ADAPTER WagoBusAdapter
  (* Standard: 61499-2; Description: Copyright (c) 2018 Jose Cabral This program and the accompanying materials are made available under the terms of the Eclipse Public License 2.0 which is available at https://www.eclipse.org/legal/epl-2.0/ SPDX-License-Identifier: EPL-2.0 *)
  (* Version 1.0, 2018-12-05, Jose Cabral *)
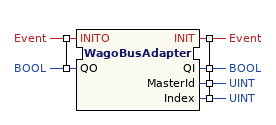
  EVENT_INPUT
    INITO WITH QO; (* Initialization Confirm *)
  END_EVENT
  EVENT_OUTPUT
    INIT WITH Index, MasterId, QI; (* Service Initialization *)
  END_EVENT
  VAR_INPUT
    QO : BOOL;
  END_VAR
  VAR_OUTPUT
    QI : BOOL;
    MasterId : UINT;
    Index : UINT;
  END_VAR
END_ADAPTER
